PROGRAM Main
VAR
	powerOn : BOOL;start : BOOL;
	reset : BOOL;
	feedbackBusy: BOOL;
	feedbackDone: BOOL;
	feedbackError: BOOL;
	feedbackErrorId: UDINT;
	feedbackAborting: BOOL;
	feedbackAborted: BOOL;
	
	errorMessage: STRING;
	errorId : UDINT;
	velocity : LREAL := 1000;

	axis1 : Axis;
	axis2 : Axis;
	nci : Nci;
	table : Table;
	feeder : Feeder(nci := nci);

	task : Task;
	state : (INIT, IDLE, RESETTING_GROUP, BUILDING_GROUP, RESETTING_FEEDER, BUILDING_TABLE, FEEDING_TABLE, MOVING, DONE, ERROR) := INIT;
	feedback : I_CommandFeedback;
END_VAR
VAR CONSTANT
	timeout : TIME := T#1S;
END_VAR

task.CyclicCall();

CASE state OF
	INIT:
		IF powerOn THEN
			powerOn := FALSE;
			axis1.EnablePositive();
			axis1.EnableNegative();
			axis1.Enable(AxisBufferMode.Aborting);
			axis2.EnablePositive();
			axis2.EnableNegative();
			axis2.Enable(AxisBufferMode.Aborting);
			IF axis1.IsReady AND axis2.IsReady THEN
				nci.ResetGroup(timeout, feedback);
				state := RESETTING_GROUP;
			END_IF
		END_IF

	RESETTING_GROUP:
		IF feedback <> 0 AND_THEN NOT feedback.Busy THEN
			IF feedback.Error THEN
				errorMessage := 'RESETTING_GROUP';
				errorId := feedback.ErrorId;
				state := ERROR;
			ELSE
				nci.BuildXYGroup(axis1, axis2, timeout, feedback);
				state := BUILDING_GROUP;
			END_IF			 
		END_IF

	BUILDING_GROUP:
		IF feedback <> 0 AND_THEN NOT feedback.Busy THEN
			IF feedback.Error THEN
				errorMessage := 'BUILDING_GROUP';
				errorId := feedback.ErrorId;
				state := ERROR;
			ELSE
				nci.SetOverride(100);
				state := IDLE;
			END_IF
		END_IF
		
	IDLE:
		IF start THEN
			start := FALSE;
			feeder.Reset(feedback);
			state := RESETTING_FEEDER;
			errorMessage := '';
			errorId := 0;
		END_IF

	RESETTING_FEEDER:		
		IF feedback <> 0 AND_THEN NOT feedback.Busy THEN
			IF feedback.Error THEN
				errorMessage := 'RESETTING_FEEDER';
				errorId := feedback.ErrorId;
				state := ERROR;
			ELSE
				state := BUILDING_TABLE;
			END_IF
		END_IF
		
	BUILDING_TABLE:
		// Method chaining with error handling
		IF table.ResetTable() THEN
			errorMessage := 'ResetTable';
			errorId := table.ErrorId;
			state := ERROR;
			RETURN;
		ELSIF table.EnableVertexSmoothing(0,
				VertexSmoothingBlendingType.PARABOLIC,
				VertexSmoothingSubType.ADAPTIVE_TOLERANCE_RADIUS,
				0.5) THEN
			errorMessage := 'EnableVertexSmoothing';
			errorId := table.ErrorId;
			state := ERROR;
			RETURN;
		ELSIF table.AddStart3D(0, 0, 0) THEN
			errorMessage := 'Start3D';
			errorId := table.ErrorId;
			state := ERROR;
			RETURN;
		ELSIF table.AddCircleOnPlane3D(
				10,
				1000, 1000, 0,
				1000, 0, 0,
				StandardPlane.XY,
				TRUE,
				velocity,
				TRUE) THEN
			errorMessage := 'AddCircleOnPlane3D';
			errorId := table.ErrorId;
			state := ERROR;
			RETURN;
		ELSIF table.End() THEN
			errorMessage := 'End';
			errorId := table.ErrorId;
			state := ERROR;
			RETURN;
		END_IF
		
		feeder.FeedTable(table, feedback);
		state := FEEDING_TABLE;		
		
	FEEDING_TABLE:
		IF feedback <> 0 AND_THEN NOT feedback.Busy THEN
			IF feedback.Error THEN
				errorMessage := 'FEEDING_TABLE';
				errorId := feedback.ErrorId;
				state := ERROR;
			ELSE
				state := MOVING;
			END_IF
		END_IF
		
	MOVING:
		IF feeder.ChannelDone THEN // end of movement
			state := DONE;
		ELSIF reset THEN
			reset := FALSE;
			state := ERROR;
		END_IF
		
	DONE:
		IF reset THEN
			reset := FALSE;
			state := IDLE;
		END_IF
		
	ERROR:
		IF reset THEN
			reset := FALSE;
			state := INIT;
		END_IF
ELSE
	state := INIT;
END_CASE

IF feedback <> 0 THEN
	feedbackBusy := feedback.Busy;
	feedbackDone := feedback.Done;
	feedbackAborted := feedback.Aborted;
	feedbackAborting := feedback.Aborting;
	feedbackError := feedback.Error;
	feedbackErrorId := feedback.ErrorId;
END_IF

END_PROGRAM

(* stored: Version 1.1.0.1, ProductVersion 3.1.4024.12
   POU Main: Id {d3d637b3-4c83-0f73-3d0f-050dde662cdf}, SpecialFunc None *)
